PROGRAM Background_Payload
VAR
	Payload_EMA		: REAL;
	Alpha			: REAL := 0.001;
	Init			: BOOL := TRUE;
	
	nBit AT %I* 	: INT;
	Voltage			: REAL;
	VoltAtEmpty		: REAL := 1.54; 
	VoltPerTon		: REAL := 1.92/70;
	Payload			: REAL;
END_VAR

Voltage	:= (INT_TO_REAL(nBit) / 32767) * 10;
Payload	:= (Voltage - VoltAtEmpty) / VoltPerTon;

IF Init THEN
	Init			:= FALSE;
	Payload_EMA 	:= Payload;
END_IF

Payload_EMA := (Alpha * Payload) + ((1 - Alpha) * Payload_EMA); //exponential mov avg

END_PROGRAM

(* stored: Version 1.1.0.1, ProductVersion 3.1.4024.6
   POU Background_Payload: Id {e111e7b3-f629-4157-80b4-b26098e5b3a4}, SpecialFunc None *)
